PROGRAM MAIN
VAR
	MyMachine : SomeMachine;
END_VAR

END_PROGRAM

(* stored: Version 1.1.0.1, ProductVersion 3.1.4024.12
   POU MAIN: Id {1ed0f9ce-8161-4573-b0c6-5057706fffd0}, SpecialFunc None *)
